(*
SPDX-FileCopyrightText: © 2026 Oleksandr Tiutyk <trofimich@gmail.com>
SPDX-License-Identifier: MIT
License: https://opensource.org/license/mit
*)

(*!
<summary>
Defines a composite automation component that acts both as a parent branch and as a child leaf in the
automation hierarchy.
</summary>
*)

INTERFACE ICompositeAutomationComponent EXTENDS
	IParentAutomationComponent,
	IChildAutomationComponent,
	IInputLeafAutomationComponent,
	IOutputLeafAutomationComponent

END_INTERFACE

(* stored: Version 1.1.0.1
   Itf ICompositeAutomationComponent: Id {be5e3b3f-f46a-4c0b-a57f-a0e8cfdaef93} *)
